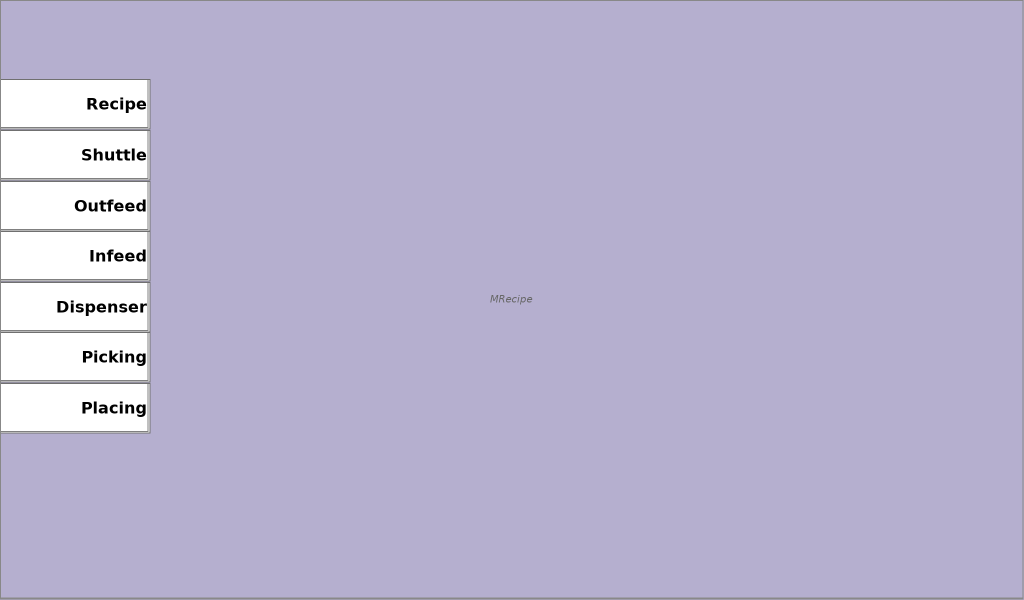
VISUALIZATION Parameter  // 1024x600
    Frame (0,0 1023x598)
        shows MRecipe()
        shows MShuttle()
        shows MOutfeed()
        shows MInfeed()
        shows MDispenser()
        shows MPicking()
        shows MPlacing()
        shows Test_Infeed()
        shows Test_Picking()
    Button (0,79 150x50), "Recipe", image: VisuSymbols.Symbols.Database2
        OnMouseDown: FrameSelectionChange Selection=SelectedFrame=5d0adf46-92b2-4ae0-bcf1-a330fcf05353, GlobSel=AssignDir=MainPage.GenElemInst_1003, AssignType=Directly, SelType=Locally
    Button (0,130 150x50), "Shuttle", image: VisuSymbols.Symbols.Database2
        OnMouseDown: FrameSelectionChange Selection=SelectedFrame=5d0adf46-92b2-4ae0-bcf1-a330fcf05353, Selection=1, GlobSel=AssignDir=MainPage.GenElemInst_1003, AssignType=Directly, SelType=Locally
    Button (0,181 150x50), "Outfeed", image: VisuSymbols.Symbols.Database2
        OnMouseDown: FrameSelectionChange Selection=SelectedFrame=5d0adf46-92b2-4ae0-bcf1-a330fcf05353, Selection=2, GlobSel=AssignDir=MainPage.GenElemInst_1003, AssignType=Directly, SelType=Locally
    Button (0,231 150x50), "Infeed", image: VisuSymbols.Symbols.Database2
        OnMouseDown: FrameSelectionChange Selection=SelectedFrame=5d0adf46-92b2-4ae0-bcf1-a330fcf05353, Selection=3, GlobSel=AssignDir=MainPage.GenElemInst_1003, AssignType=Directly, SelType=Locally
    Button (0,282 150x50), "Dispenser", image: VisuSymbols.Symbols.Database2
        OnMouseDown: FrameSelectionChange Selection=SelectedFrame=5d0adf46-92b2-4ae0-bcf1-a330fcf05353, Selection=4, GlobSel=AssignDir=MainPage.GenElemInst_1003, AssignType=Directly, SelType=Locally
    Button (0,332 150x50), "Picking", image: VisuSymbols.Symbols.Database2
        OnMouseDown: FrameSelectionChange Selection=SelectedFrame=5d0adf46-92b2-4ae0-bcf1-a330fcf05353, Selection=5, GlobSel=AssignDir=MainPage.GenElemInst_1003, AssignType=Directly, SelType=Locally
    Button (0,383 150x50), "Placing", image: VisuSymbols.Symbols.Database2
        OnMouseDown: FrameSelectionChange Selection=SelectedFrame=5d0adf46-92b2-4ae0-bcf1-a330fcf05353, Selection=6, GlobSel=AssignDir=MainPage.GenElemInst_1003, AssignType=Directly, SelType=Locally
END_VISUALIZATION

(* stored: Version 1.1.0.1, ProductVersion 3.1.4024.12
   Visu Parameter: Id {88167398-2cef-4608-9ef8-04b25a7a5719} *)
